//{attribute 'qualified_only'}
VAR_GLOBAL

	// Motor axes
    {attribute 'pytmc' := 'pv: CRIX:DPL:MMS:X'}
    {attribute 'TcLinkTo' := '.bLimitForwardEnable  := TIID^Device 1 (EtherCAT)^Term 5 (EK1200)^Term 6 (EK1122-0080)^DRL02-EK0 (EK1101-0080)^DRL02-E1 (EL7031)^STM Status^Status^Digital input 2;
                              .bLimitBackwardEnable := TIID^Device 1 (EtherCAT)^Term 5 (EK1200)^Term 6 (EK1122-0080)^DRL02-EK0 (EK1101-0080)^DRL02-E1 (EL7031)^STM Status^Status^Digital input 1'}
	M1 : DUT_MotionStage := (bPowerSelf:=TRUE, nEnableMode:=ENUM_StageEnableMode.ALWAYS);
	//stDPXMotor : DUT_MotionStage;
	
	{attribute 'pytmc' := 'pv: CRIX:DPL:MMS:Y'}
    {attribute 'TcLinkTo' := '.bLimitForwardEnable  := TIID^Device 1 (EtherCAT)^Term 5 (EK1200)^Term 6 (EK1122-0080)^DRL02-EK0 (EK1101-0080)^DRL02-E3 (EL7031)^STM Status^Status^Digital input 1;
                              .bLimitBackwardEnable := TIID^Device 1 (EtherCAT)^Term 5 (EK1200)^Term 6 (EK1122-0080)^DRL02-EK0 (EK1101-0080)^DRL02-E3 (EL7031)^STM Status^Status^Digital input 2'}
	M2 : DUT_MotionStage := (bPowerSelf:=TRUE, nEnableMode:=ENUM_StageEnableMode.ALWAYS);
	//stDPYMotor : DUT_MotionStage;
	
	{attribute 'pytmc' := 'pv: CRIX:DPL:MMS:Z'}
    {attribute 'TcLinkTo' := '.bLimitForwardEnable  := TIID^Device 1 (EtherCAT)^Term 5 (EK1200)^Term 6 (EK1122-0080)^DRL02-EK0 (EK1101-0080)^DRL02-E4 (EL7031)^STM Status^Status^Digital input 1;
                              .bLimitBackwardEnable := TIID^Device 1 (EtherCAT)^Term 5 (EK1200)^Term 6 (EK1122-0080)^DRL02-EK0 (EK1101-0080)^DRL02-E4 (EL7031)^STM Status^Status^Digital input 2'}
	M3 : DUT_MotionStage :=(bPowerSelf:=TRUE,nEnableMode:=ENUM_StageEnableMode.ALWAYS);
	//stDPZMotor : DUT_MotionStage;
	
	
	
	
    {attribute 'pytmc' := 'pv: CRIX:OBJ:MMS:X'}
	{attribute 'TcLinkTo' := '.bLimitForwardEnable  := TIID^Device 1 (EtherCAT)^Term 5 (EK1200)^Term 6 (EK1122-0080)^DRL02-EK0 (EK1101-0080)^DRL02-E6 (EL7031)^STM Status^Status^Digital input 2;
                              .bLimitBackwardEnable := TIID^Device 1 (EtherCAT)^Term 5 (EK1200)^Term 6 (EK1122-0080)^DRL02-EK0 (EK1101-0080)^DRL02-E6 (EL7031)^STM Status^Status^Digital input 1'}
	M4: DUT_MotionStage :=(bPowerSelf:=TRUE ,nEnableMode:=ENUM_StageEnableMode.ALWAYS);
	//stOBJXMotor : DUT_MotionStage;
	
	{attribute 'pytmc' := 'pv: CRIX:OBJ:MMS:Y'}
	{attribute 'TcLinkTo' := '.bLimitForwardEnable  := TIID^Device 1 (EtherCAT)^Term 5 (EK1200)^Term 6 (EK1122-0080)^DRL02-EK0 (EK1101-0080)^DRL02-E7 (EL7031)^STM Status^Status^Digital input 1;
                              .bLimitBackwardEnable := TIID^Device 1 (EtherCAT)^Term 5 (EK1200)^Term 6 (EK1122-0080)^DRL02-EK0 (EK1101-0080)^DRL02-E7 (EL7031)^STM Status^Status^Digital input 2'}
	M5 : DUT_MotionStage :=(bPowerSelf:=TRUE, nEnableMode:=ENUM_StageEnableMode.ALWAYS);
	//stOBJYMotor : DUT_MotionStage;
	
	{attribute 'pytmc' := 'pv: CRIX:OBJ:MMS:Z'}
	{attribute 'TcLinkTo' := '.bLimitForwardEnable  := TIID^Device 1 (EtherCAT)^Term 5 (EK1200)^Term 6 (EK1122-0080)^DRL02-EK0 (EK1101-0080)^DRL02-E9 (EL7031)^STM Status^Status^Digital input 1;
                              .bLimitBackwardEnable := TIID^Device 1 (EtherCAT)^Term 5 (EK1200)^Term 6 (EK1122-0080)^DRL02-EK0 (EK1101-0080)^DRL02-E9 (EL7031)^STM Status^Status^Digital input 2'}
	M6 : DUT_MotionStage :=(bPowerSelf:=TRUE, nEnableMode:=ENUM_StageEnableMode.ALWAYS);
	//stOBJZMotor : DUT_MotionStage;

	
	
	{attribute 'pytmc' := 'pv: CRIX:PDET:MMS:Y'}
    {attribute 'TcLinkTo' := '.bLimitForwardEnable  := TIID^Device 1 (EtherCAT)^Term 5 (EK1200)^Term 6 (EK1122-0080)^DRL02-EK0 (EK1101-0080)^DRL02-E11 (EL7031)^STM Status^Status^Digital input 1;
                              .bLimitBackwardEnable := TIID^Device 1 (EtherCAT)^Term 5 (EK1200)^Term 6 (EK1122-0080)^DRL02-EK0 (EK1101-0080)^DRL02-E11 (EL7031)^STM Status^Status^Digital input 2'}	
	M7 : DUT_MotionStage := (bPowerSelf:=TRUE, nEnableMode:=ENUM_StageEnableMode.ALWAYS);
	//stPDYMotor : DUT_MotionStage;	
	{attribute 'pytmc' := 'pv: CRIX:PDET:MMS:THETA'}
    {attribute 'TcLinkTo' := '.bLimitForwardEnable  := TIID^Device 1 (EtherCAT)^Term 5 (EK1200)^Term 6 (EK1122-0080)^DRL02-EK0 (EK1101-0080)^DRL02-E13 (EL7041)^STM Status^Status^Digital input 1;
                              .bLimitBackwardEnable := TIID^Device 1 (EtherCAT)^Term 5 (EK1200)^Term 6 (EK1122-0080)^DRL02-EK0 (EK1101-0080)^DRL02-E13 (EL7041)^STM Status^Status^Digital input 2'}
	M8 : DUT_MotionStage := (bPowerSelf:=TRUE);
	//stPDRotMotor : DUT_MotionStage;
	
	M9 : DUT_MotionStage;
	//stILMXMotor : DUT_MotionStage;
	M10 : DUT_MotionStage;
	//stILMYMotor : DUT_MotionStage;
	M11 : DUT_MotionStage;
	//stILMZMotor : DUT_MotionStage;

	{attribute 'pytmc' := 'pv: CRIX:QSTR:MMS:X'}
    {attribute 'TcLinkTo' := '.bLimitForwardEnable  := TIID^Device 1 (EtherCAT)^Term 5 (EK1200)^Term 6 (EK1122-0080)^DRL02-EK0 (EK1101-0080)^DRL02-E17 (EL7031)^STM Status^Status^Digital input 1;
                              .bLimitBackwardEnable := TIID^Device 1 (EtherCAT)^Term 5 (EK1200)^Term 6 (EK1122-0080)^DRL02-EK0 (EK1101-0080)^DRL02-E17 (EL7031)^STM Status^Status^Digital input 2'}
	M12 : DUT_MotionStage := (bPowerSelf:=TRUE);
	//stQSTXMotor : DUT_MotionStage;
	{attribute 'pytmc' := 'pv: CRIX:QSTR:MMS:Y'}
    {attribute 'TcLinkTo' := '.bLimitForwardEnable  := TIID^Device 1 (EtherCAT)^Term 5 (EK1200)^Term 6 (EK1122-0080)^DRL02-EK0 (EK1101-0080)^DRL02-E19 (EL7031)^STM Status^Status^Digital input 1;
                              .bLimitBackwardEnable := TIID^Device 1 (EtherCAT)^Term 5 (EK1200)^Term 6 (EK1122-0080)^DRL02-EK0 (EK1101-0080)^DRL02-E19 (EL7031)^STM Status^Status^Digital input 2'}
	M13 : DUT_MotionStage := (bPowerSelf:=TRUE);
	//stQSTYMotor : DUT_MotionStage;
	
	M14 : DUT_MotionStage; // Cryopump 1
	M15 : DUT_MotionStage; // Cryopump 2
	
	{attribute 'pytmc' := 'pv: CRIX:SDS:MMS:X'}
	{attribute 'TcLinkTo' := '.bLimitForwardEnable := TIID^Device 1 (EtherCAT)^Term 5 (EK1200)^Term 6 (EK1122-0080)^DRL02-EK0 (EK1101-0080)^Term 82 (EL1084)^Channel 1^Input;
							 '.bLimBackwardEnable := TIID^Device 1 (EtherCAT)^Term 5 (EK1200)^Term 6 (EK1122-0080)^DRL02-EK0 (EK1101-0080)^Term 82 (EL1084)^Channel 2^Input'}
	M16 : DUT_MotionStage := (bPowerSelf:=TRUE, nEnableMode:=ENUM_StageEnableMode.DURING_MOTION); //stSDSXMotor : DUT_MotionStage;
	
	{attribute 'pytmc' := 'pv: CRIX:SDS:MMS:Y'}
	{attribute 'TcLinkTo' := '.bLimitForwardEnable := TIID^Device 1 (EtherCAT)^Term 5 (EK1200)^Term 6 (EK1122-0080)^DRL02-EK0 (EK1101-0080)^DRL02-E26 (EL7031)^STM Status^Status^Digital input 1;
							 '.bLimBackwardEnable := TIID^Device 1 (EtherCAT)^Term 5 (EK1200)^Term 6 (EK1122-0080)^DRL02-EK0 (EK1101-0080)^DRL02-E26 (EL7031)^STM Status^Status^Digital input 2'}
	M17 : DUT_MotionStage := (bPowerSelf:=TRUE, nEnableMode:=ENUM_StageEnableMode.DURING_MOTION); //stSDSYMotor : DUT_MotionStage;
	
	{attribute 'pytmc' := 'pv: CRIX:SDS:MMS:Z'}
	{attribute 'TcLinkTo' := '.bLimitForwardEnable := TIID^Device 1 (EtherCAT)^Term 5 (EK1200)^Term 6 (EK1122-0080)^DRL02-EK0 (EK1101-0080)^DRL02-E27 (EL7031)^STM Status^Status^Digital input 1;
							 '.bLimBackwardEnable := TIID^Device 1 (EtherCAT)^Term 5 (EK1200)^Term 6 (EK1122-0080)^DRL02-EK0 (EK1101-0080)^DRL02-E27 (EL7031)^STM Status^Status^Digital input 2'}
	M18 : DUT_MotionStage := (bPowerSelf:=TRUE, nEnableMode:=ENUM_StageEnableMode.DURING_MOTION); //stSDSZMotor : DUT_MotionStage;
	
	{attribute 'pytmc' := 'pv: CRIX:SDS:MMS:RY'}
(*	{attribute 'TcLinkTo' := '.bLimitForwardEnable := ;   // There are currently no limits on this stage
							 '.bLimBackwardEnable := '} *)
	M19 : DUT_MotionStage := (bPowerSelf:=TRUE, nEnableMode:=ENUM_StageEnableMode.DURING_MOTION); //stSDSRotMotor : DUT_MotionStage;
	
	{attribute 'pytmc' := 'pv: CRIX:SDS:MMS:SHROUD'}
(*	{attribute 'TcLinkTo' := '.bLimitForwardEnable := ;  // There are currently no limits on this stage
							 '.bLimBackwardEnable := '} *)
	M20 : DUT_MotionStage := (bPowerSelf:=TRUE, nEnableMode:=ENUM_StageEnableMode.DURING_MOTION); //stSDSShroudMotor : DUT_MotionStage;
	
    {attribute 'pytmc' := 'pv: CRIX:CRYO:MMS:X'}
    {attribute 'TcLinkTo' := '.bLimitForwardEnable  := TIID^Device 1 (EtherCAT)^Term 5 (EK1200)^Term 6 (EK1122-0080)^DRL02-EK0 (EK1101-0080)^DRL02-ECJ1 (EK1122)^CryoStat (EK1101)^Cryo X (EL7041)^STM Status^Status^Digital input 1;
                              .bLimitBackwardEnable := TIID^Device 1 (EtherCAT)^Term 5 (EK1200)^Term 6 (EK1122-0080)^DRL02-EK0 (EK1101-0080)^DRL02-ECJ1 (EK1122)^CryoStat (EK1101)^Cryo X (EL7041)^STM Status^Status^Digital input 2'}
    M22 : DUT_MotionStage := (bPowerSelf:=TRUE, nEnableMode:=ENUM_StageEnableMode.ALWAYS); //CryoStat X
    {attribute 'pytmc' := 'pv: CRIX:CRYO:MMS:Y'}
    {attribute 'TcLinkTo' := '.bLimitForwardEnable  := TIID^Device 1 (EtherCAT)^Term 5 (EK1200)^Term 6 (EK1122-0080)^DRL02-EK0 (EK1101-0080)^DRL02-ECJ1 (EK1122)^CryoStat (EK1101)^Cryo Y (EL7041)^STM Status^Status^Digital input 1;
                              .bLimitBackwardEnable := TIID^Device 1 (EtherCAT)^Term 5 (EK1200)^Term 6 (EK1122-0080)^DRL02-EK0 (EK1101-0080)^DRL02-ECJ1 (EK1122)^CryoStat (EK1101)^Cryo Y (EL7041)^STM Status^Status^Digital input 2'}
    M23 : DUT_MotionStage := (bPowerSelf:=TRUE, nEnableMode:=ENUM_StageEnableMode.ALWAYS); //CryoStat Y
    {attribute 'pytmc' := 'pv: CRIX:CRYO:MMS:Z'}
    {attribute 'TcLinkTo' := '.bLimitForwardEnable  := TIID^Device 1 (EtherCAT)^Term 5 (EK1200)^Term 6 (EK1122-0080)^DRL02-EK0 (EK1101-0080)^DRL02-ECJ1 (EK1122)^CryoStat (EK1101)^Cryo Z (EL7041)^STM Status^Status^Digital input 1;
                              .bLimitBackwardEnable := TIID^Device 1 (EtherCAT)^Term 5 (EK1200)^Term 6 (EK1122-0080)^DRL02-EK0 (EK1101-0080)^DRL02-ECJ1 (EK1122)^CryoStat (EK1101)^Cryo Z (EL7041)^STM Status^Status^Digital input 2'}
    M24 : DUT_MotionStage:= (bPowerSelf:=TRUE, nEnableMode:=ENUM_StageEnableMode.ALWAYS); //CryoStat Z
    {attribute 'pytmc' := 'pv: CRIX:CRYO:MMS:RY'}
    M25 : DUT_MotionStage := (bPowerSelf:=TRUE, nEnableMode:=ENUM_StageEnableMode.ALWAYS); //CryoStat rY
     {attribute 'pytmc' := 'pv: CRIX:RCI:MMS:X'}
     {attribute 'TcLinkTo' := '.bLimitForwardEnable  := TIID^Device 1 (EtherCAT)^Term 5 (EK1200)^Term 6 (EK1122-0080)^DRL02-EK0 (EK1101-0080)^DRL02-ECJ0 (EK1122-0080)^RCI (EK1101-0080)^RCI X (EL7041)^STM Status^Status^Digital input 1;
                              .bLimitBackwardEnable := TIID^Device 1 (EtherCAT)^Term 5 (EK1200)^Term 6 (EK1122-0080)^DRL02-EK0 (EK1101-0080)^DRL02-ECJ0 (EK1122-0080)^RCI (EK1101-0080)^RCI X (EL7041)^STM Status^Status^Digital input 2'}
    M26 : DUT_MotionStage := (bPowerSelf:=TRUE, nEnableMode:=ENUM_StageEnableMode.ALWAYS); //RCI X
     {attribute 'pytmc' := 'pv: CRIX:RCI:MMS:Y'}
     {attribute 'TcLinkTo' := '.bLimitForwardEnable  := TIID^Device 1 (EtherCAT)^Term 5 (EK1200)^Term 6 (EK1122-0080)^DRL02-EK0 (EK1101-0080)^DRL02-ECJ0 (EK1122-0080)^RCI (EK1101-0080)^RCI Y (EL7041)^STM Status^Status^Digital input 1;
                              .bLimitBackwardEnable := TIID^Device 1 (EtherCAT)^Term 5 (EK1200)^Term 6 (EK1122-0080)^DRL02-EK0 (EK1101-0080)^DRL02-ECJ0 (EK1122-0080)^RCI (EK1101-0080)^RCI Y (EL7041)^STM Status^Status^Digital input 2'}
    M27 : DUT_MotionStage := (bPowerSelf:=TRUE, nEnableMode:=ENUM_StageEnableMode.ALWAYS); //RCI Y
     {attribute 'pytmc' := 'pv: CRIX:RCI:MMS:Z'}
     {attribute 'TcLinkTo' := '.bLimitForwardEnable  := TIID^Device 1 (EtherCAT)^Term 5 (EK1200)^Term 6 (EK1122-0080)^DRL02-EK0 (EK1101-0080)^DRL02-ECJ0 (EK1122-0080)^RCI (EK1101-0080)^RCI Z (EL7041)^STM Status^Status^Digital input 1;
                              .bLimitBackwardEnable := TIID^Device 1 (EtherCAT)^Term 5 (EK1200)^Term 6 (EK1122-0080)^DRL02-EK0 (EK1101-0080)^DRL02-ECJ0 (EK1122-0080)^RCI (EK1101-0080)^RCI Z (EL7041)^STM Status^Status^Digital input 2'}
    M28 : DUT_MotionStage := (bPowerSelf:=TRUE, nEnableMode:=ENUM_StageEnableMode.ALWAYS); //RCI Z
     {attribute 'pytmc' := 'pv: CRIX:RCI:MMS:RX'}
    M29 : DUT_MotionStage := (bPowerSelf:=TRUE, nEnableMode:=ENUM_StageEnableMode.ALWAYS); //RCI rX
     {attribute 'pytmc' := 'pv: CRIX:BEAM:MMS:X'}
     {attribute 'TcLinkTo' := '.bLimitForwardEnable  := TIID^Device 1 (EtherCAT)^Term 5 (EK1200)^Term 6 (EK1122-0080)^DRL02-EK0 (EK1101-0080)^DRL02-ECJ0 (EK1122-0080)^Term 113 (EK1101-0080)^Beamblock X (EL7041)^STM Status^Status^Digital input 1;
                              .bLimitBackwardEnable := TIID^Device 1 (EtherCAT)^Term 5 (EK1200)^Term 6 (EK1122-0080)^DRL02-EK0 (EK1101-0080)^DRL02-ECJ0 (EK1122-0080)^Term 113 (EK1101-0080)^Beamblock X (EL7041)^STM Status^Status^Digital input 2'}
    M30 : DUT_MotionStage := (bPowerSelf:=TRUE, nEnableMode:=ENUM_StageEnableMode.ALWAYS); //BEAM X
     {attribute 'pytmc' := 'pv: CRIX:BEAM:MMS:Y'}
     {attribute 'TcLinkTo' := '.bLimitForwardEnable  := TIID^Device 1 (EtherCAT)^Term 5 (EK1200)^Term 6 (EK1122-0080)^DRL02-EK0 (EK1101-0080)^DRL02-ECJ0 (EK1122-0080)^Term 113 (EK1101-0080)^Beamblock Y (EL7041)^STM Status^Status^Digital input 1;
                              .bLimitBackwardEnable := TIID^Device 1 (EtherCAT)^Term 5 (EK1200)^Term 6 (EK1122-0080)^DRL02-EK0 (EK1101-0080)^DRL02-ECJ0 (EK1122-0080)^Term 113 (EK1101-0080)^Beamblock Y (EL7041)^STM Status^Status^Digital input 2'}
    M31 : DUT_MotionStage := (bPowerSelf:=TRUE, nEnableMode:=ENUM_StageEnableMode.ALWAYS); //BEAM Y
     {attribute 'pytmc' := 'pv: CRIX:BEAM:MMS:Z'}
     {attribute 'TcLinkTo' := '.bLimitForwardEnable  := TIID^Device 1 (EtherCAT)^Term 5 (EK1200)^Term 6 (EK1122-0080)^DRL02-EK0 (EK1101-0080)^DRL02-ECJ0 (EK1122-0080)^Term 113 (EK1101-0080)^Beamblock Z (EL7041)^STM Status^Status^Digital input 1;
                              .bLimitBackwardEnable := TIID^Device 1 (EtherCAT)^Term 5 (EK1200)^Term 6 (EK1122-0080)^DRL02-EK0 (EK1101-0080)^DRL02-ECJ0 (EK1122-0080)^Term 113 (EK1101-0080)^Beamblock Z (EL7041)^STM Status^Status^Digital input 2'}
    M32 : DUT_MotionStage := (bPowerSelf:=TRUE, nEnableMode:=ENUM_StageEnableMode.ALWAYS); //BEAM Z
     {attribute 'pytmc' := 'pv: CRIX:CAM:MMS:X'}
     {attribute 'TcLinkTo' := '.bLimitForwardEnable  := TIID^Device 1 (EtherCAT)^Term 5 (EK1200)^Term 6 (EK1122-0080)^DRL02-EK0 (EK1101-0080)^DRL02-ECJ0 (EK1122-0080)^Term 109 (EK1101-0080)^Camera X (EL7041)^STM Status^Status^Digital input 1;
                              .bLimitBackwardEnable := TIID^Device 1 (EtherCAT)^Term 5 (EK1200)^Term 6 (EK1122-0080)^DRL02-EK0 (EK1101-0080)^DRL02-ECJ0 (EK1122-0080)^Term 109 (EK1101-0080)^Camera X (EL7041)^STM Status^Status^Digital input 2'}
    M33 : DUT_MotionStage := (bPowerSelf:=TRUE, nEnableMode:=ENUM_StageEnableMode.ALWAYS); //CAM X
     {attribute 'pytmc' := 'pv: CRIX:CAM:MMS:Y'}
     {attribute 'TcLinkTo' := '.bLimitForwardEnable  := TIID^Device 1 (EtherCAT)^Term 5 (EK1200)^Term 6 (EK1122-0080)^DRL02-EK0 (EK1101-0080)^DRL02-ECJ0 (EK1122-0080)^Term 109 (EK1101-0080)^Camera Y (EL7041)^STM Status^Status^Digital input 1;
                              .bLimitBackwardEnable := TIID^Device 1 (EtherCAT)^Term 5 (EK1200)^Term 6 (EK1122-0080)^DRL02-EK0 (EK1101-0080)^DRL02-ECJ0 (EK1122-0080)^Term 109 (EK1101-0080)^Camera Y (EL7041)^STM Status^Status^Digital input 2'}
    M34 : DUT_MotionStage := (bPowerSelf:=TRUE, nEnableMode:=ENUM_StageEnableMode.ALWAYS); //CAM Z
     {attribute 'pytmc' := 'pv: CRIX:OUTCOUP:MMS:Y'}
     {attribute 'TcLinkTo' := '.bLimitForwardEnable  := TIID^Device 1 (EtherCAT)^Term 5 (EK1200)^Term 6 (EK1122-0080)^DRL02-EK0 (EK1101-0080)^DRL02-E31 (EL7031)^STM Status^Status^Digital input 1;
                              .bLimitBackwardEnable := TIID^Device 1 (EtherCAT)^Term 5 (EK1200)^Term 6 (EK1122-0080)^DRL02-EK0 (EK1101-0080)^DRL02-E31 (EL7031)^STM Status^Status^Digital input 2'}
    M35 : DUT_MotionStage := (bPowerSelf:=TRUE, nEnableMode:=ENUM_StageEnableMode.ALWAYS); //OUTCOUP LENS Y
    
(*	
	M21 : DUT_MotionStage; // Out-coupling y
 *)
 
 (* not needed for now; it has a manual knob
 // NOTE: Questar is M21, even though Outcoupling Y stage is before it on the DIN rail
 	{attribute 'pytmc' := 'pv: CRIX:QSTR:MMS:FOCUS'}
    {attribute 'TcLinkTo' := '.bLimitForwardEnable  := TIID^Device 1 (EtherCAT)^Term 5 (EK1200)^Term 6 (EK1122-0080)^DRL02-EK0 (EK1101-0080)^DRL02-E33 (EL7031)^STM Status^Status^Digital input 1;
                              .bLimitBackwardEnable := TIID^Device 1 (EtherCAT)^Term 5 (EK1200)^Term 6 (EK1122-0080)^DRL02-EK0 (EK1101-0080)^DRL02-E33 (EL7031)^STM Status^Status^Digital input 2'}
	M21 : DUT_MotionStage; // Questar Focus
*)
	//Catcher Axes
	 {attribute 'pytmc' := 'pv: CRIX:RCC:MMS:X'}
     {attribute 'TcLinkTo' := '.bLimitForwardEnable  := TIIB[Catcher_E1_EL7041]^STM Status^Status^Digital input 2;
                              .bLimitBackwardEnable := TIIB[Catcher_E1_EL7041]^STM Status^Status^Digital input 1'}
    M37 : DUT_MotionStage := (bPowerSelf:=TRUE, nEnableMode:=ENUM_StageEnableMode.ALWAYS); //RCC X
     {attribute 'pytmc' := 'pv: CRIX:RCC:MMS:Y'}
	 {attribute 'TcLinkTo' := '.bLimitForwardEnable  := TIIB[Catcher_E3_EL7041]^STM Status^Status^Digital input 1;
                              .bLimitBackwardEnable := TIIB[Catcher_E3_EL7041]^STM Status^Status^Digital input 2'}
    M38 : DUT_MotionStage := (bPowerSelf:=TRUE, nEnableMode:=ENUM_StageEnableMode.ALWAYS); //RCC Y
     {attribute 'pytmc' := 'pv: CRIX:RCC:MMS:Z'}
     {attribute 'TcLinkTo' := '.bLimitForwardEnable  := TIIB[Catcher_E4_EL7041]^STM Status^Status^Digital input 2;
                              .bLimitBackwardEnable := TIIB[Catcher_E4_EL7041]^STM Status^Status^Digital input 1'}
    M39 : DUT_MotionStage := (bPowerSelf:=TRUE, nEnableMode:=ENUM_StageEnableMode.ALWAYS); //RCC Z
    
	 // VLS SLIT TOP
	{attribute 'TcLinkTo' := '	.bLimitForwardEnable:=TIIB[VLS_EP6_EP7041-1002]^STM Status^Status^Digital input 1;
								.bLimitBackwardEnable:=TIIB[VLS_EP6_EP7041-1002]^STM Status^Status^Digital input 2'}
    {attribute 'pytmc' := '
        pv: CRIX:VLS:MMS:SLTOP
        field: DESC VLS Slit TOP Blade
    '}
    M40: DUT_MotionStage;

	 // VLS SLIT BOTTOM
	{attribute 'TcLinkTo' := '	.bLimitForwardEnable:=TIIB[VLS_EP7_EP7041-1002]^STM Status^Status^Digital input 1;
								.bLimitBackwardEnable:=TIIB[VLS_EP7_EP7041-1002]^STM Status^Status^Digital input 2'}
    {attribute 'pytmc' := '
        pv: CRIX:VLS:MMS:SLBOTTOM
        field: DESC VLS Slit BOTTOM Blade
    '}
    M41: DUT_MotionStage;
	
	// VLS SLIT RIGHT
	{attribute 'TcLinkTo' := '	.bLimitForwardEnable:=TIIB[VLS_EP8_EP7041-1002]^STM Status^Status^Digital input 1;
								.bLimitBackwardEnable:=TIIB[VLS_EP8_EP7041-1002]^STM Status^Status^Digital input 2'}
    {attribute 'pytmc' := '
        pv: CRIX:VLS:MMS:SLRIGHT
        field: DESC VLS Slit RIGHT Blade
    '}
    M42: DUT_MotionStage;
	
	
	// VLS SLIT LEFT
	{attribute 'TcLinkTo' := '	.bLimitForwardEnable:=TIIB[VLS_EP9_EP7041-1002]^STM Status^Status^Digital input 1;
								.bLimitBackwardEnable:=TIIB[VLS_EP9_EP7041-1002]^STM Status^Status^Digital input 2'}
    {attribute 'pytmc' := '
        pv: CRIX:VLS:MMS:SLLEFT
        field: DESC VLS Slit LEFT Blade
    '}
    M43: DUT_MotionStage;
	
	
	
	// VLS focusing mirror pitch
	{attribute 'TcLinkTo' := '	.bLimitForwardEnable:=TIIB[VLS_EP10_EP7041-3102]^STM Status^Status^Digital input 2;
								.bLimitBackwardEnable:=TIIB[VLS_EP10_EP7041-3102]^STM Status^Status^Digital input 1;
								.nRawEncoderUINT:=TIIB[VLS_EP10_EP7041-3102]^ENC Status compact^Counter value;
								.bHome:=TIIB[VLS_EP10_EP7041-3102]^ENC Status compact^Status^Status of input C'}
    {attribute 'pytmc' := '
        pv:  CRIX:VLS:MMS:MP
        field: DESC VLS Focus Mirror Pitch
    '}
    M44: DUT_MotionStage;
	
	// VLS grating pitch
	{attribute 'TcLinkTo' := '	.bLimitForwardEnable:=TIIB[VLS_EP11_EP7041-3102]^STM Status^Status^Digital input 2;
								.bLimitBackwardEnable:=TIIB[VLS_EP11_EP7041-3102]^STM Status^Status^Digital input 1;
								.nRawEncoderUINT:=TIIB[VLS_EP11_EP7041-3102]^ENC Status compact^Counter value;
								.bHome:=TIIB[VLS_EP11_EP7041-3102]^ENC Status compact^Status^Status of input C'}
    {attribute 'pytmc' := '
        pv:  CRIX:VLS:MMS:GP
        field: DESC VLS Grating Pitch
    '}
    M45: DUT_MotionStage;
	
	// VLS camera Pitch
	{attribute 'TcLinkTo' := '	.bLimitForwardEnable:=TIIB[VLS_EP12_EP7041-3102]^STM Status^Status^Digital input 1;
								.bLimitBackwardEnable:=TIIB[VLS_EP12_EP7041-3102]^STM Status^Status^Digital input 2;
								.bHome:=TIIB[VLS_EP12_EP7041-3102]^ENC Status compact^Status^Status of input C'}
    {attribute 'pytmc' := '
        pv: CRIX:VLS:CAM:MMS:PITCH
        field: DESC VLS Camera Pitch
    '}
    M46: DUT_MotionStage;
	
	// VLS camera Distance
	{attribute 'TcLinkTo' := '	.bLimitForwardEnable:=TIIB[VLS_EP13_EP7041-3102]^STM Status^Status^Digital input 2;
								.bLimitBackwardEnable:=TIIB[VLS_EP13_EP7041-3102]^STM Status^Status^Digital input 1;
								.bHome:=TIIB[VLS_EP13_EP7041-3102]^ENC Status compact^Status^Status of input C'}
    {attribute 'pytmc' := '
        pv:  CRIX:VLS:CAM:MMS:DIST
        field: DESC VLS Camera Translation
    '}
    M47: DUT_MotionStage;
END_VAR

(* stored: Version 1.1.0.1, ProductVersion 3.1.4022.18
   GVL Main: Id {743c36cb-e5dd-4408-91ed-5169699d82d2} *)
